SUBAPPLICATION Versuch_407 (* Versuch Array Summe *)
  (* Standard: 61499-2; Description: Copyright (c) 2023 Meisterschulen am Ostbahnhof This program and the accompanying materials are made available under the terms of the Eclipse Public License 2.0 which is available at https://www.eclipse.org/legal/epl-2.0/ SPDX-License-Identifier: EPL-2.0 *)
  (* Version 1.0, 2023-10-23, Franz Höpfinger, Meisterschulen am Ostbahnhof *)
  PACKAGE Versuche;
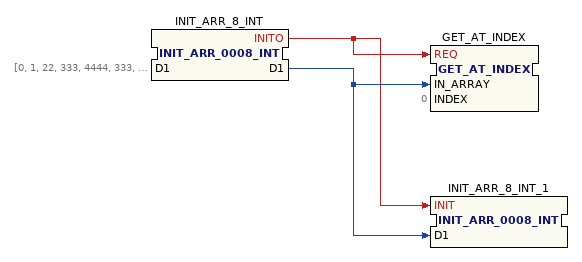
  FBS
    INIT_ARR_8_INT : logiBUS::utils::generate::INIT_ARR_0008_INT(D1 := [0, 1, 22, 333, 4444, 333, 22, 1]);
    GET_AT_INDEX : eclipse4diac::convert::GET_AT_INDEX(INDEX := 0);
    INIT_ARR_8_INT_1 : logiBUS::utils::generate::INIT_ARR_0008_INT;
  END_FBS
  EVENT_CONNECTIONS
    INIT_ARR_8_INT.INITO TO GET_AT_INDEX.REQ;
    INIT_ARR_8_INT.INITO TO INIT_ARR_8_INT_1.INIT;
  END_CONNECTIONS
  DATA_CONNECTIONS
    INIT_ARR_8_INT.D1 TO GET_AT_INDEX.IN_ARRAY;
    INIT_ARR_8_INT.D1 TO INIT_ARR_8_INT_1.D1;
  END_CONNECTIONS
END_SUBAPPLICATION
